PROGRAM MAIN
VAR
	
	// general use variables
	bLocalVar_1				: BOOL;
	bActivateTimeout		: BOOL;
	bHighLevelAlarm			: BOOL;
	bLowLevelAlarm			: BOOL;
	nRetryCounter			: USINT;
	tTotalCycleTime 		: TIME;
	tTimeoutTime			: TIME;
	sMachineState			: STRING(30);
	sPrevMachineState		: STRING(30);
	sErrorMsg				: STRING(50);
	tmrProcessTimer			: Tc2_Standard.TON;
	
	// function block and interface definitions
	fbFurnace 				: FB_Furnace;
	fbGantry 				: FB_Gantry;
	fbQuenchTank 			: FB_QuenchTank;
	fbRecipie				: FB_Recipe;
	fbAlarmManager			: FB_AlarmManager;
	fbTimeout				: FB_Timeout;
	fbStackLight			: FB_StackLight;
	iGantry					: I_Gantry;
	
	// recipe variables
	bCreateRecipe			: BOOL;
	bEditRecipe         	: BOOL;
	bDeleteRecipe			: BOOL;
	tHeatSetTime			: TIME;
	tQuenchTime				: TIME;
	sRecipeName				: STRING(20);
	
	// salt furnace variables
	bSaltCoverOn	    	: BOOL;	
	
	// quench tank variables

END_VAR

// *** GANTRY CONTROL ********************************************************************************

IF sMachineState = 'Startup' THEN
	sMachineState := 'Navigating Home';
	
ELSIF sMachineState = 'Idle' THEN
	sPrevMachineState := 'Idle';

ELSIF sMachineState = 'Navigating to Start Position' THEN
	IF sPrevMachineState <> 'Navigating to Start Position' THEN
		sPrevMachineState := 'Navigating to Start Position';
		iGantry.M_GoPreHeatSet();
		fbTimeout(bActivate := FALSE);
		bActivateTimeout := TRUE;
		tTimeoutTime := T#20S;
		nRetryCounter := 0;
	END_IF

	IF iGantry.M_GetPosition() = 'pre heat set' THEN
		sMachineState := 'Waiting for Start';
	ELSIF fbTimeout.nAttempts >= 3 THEN
		sMachineState := 'Help Required';
		sErrorMsg := 'Unable to move to start pos from home';
	ELSIF fbTimeout.nAttempts > nRetryCounter THEN
		iGantry.M_GoPreHeatSet();
		nRetryCounter := nRetryCounter + 1;
	END_IF

ELSIF sMachineState = 'Waiting for Start' THEN
    RETURN;
	
ELSIF sMachineState = 'Getting Salty' THEN
	IF sPrevMachineState <> 'Getting Salty' THEN
		sPrevMachineState := 'Getting Salty';
	    iGantry.M_GoHeatSet();
		fbTimeout(bActivate := FALSE);
		bActivateTimeout := TRUE;
		tTimeoutTime := T#10S;
		nRetryCounter := 0;
	END_IF

	IF iGantry.M_GetPosition() = 'setting shape' THEN
		sMachineState := 'Heat Soaking';
	ELSIF fbTimeout.nAttempts >= 3 THEN
		sMachineState := 'Help Required';
		sErrorMsg := 'Unable to enter salt bath';
	ELSIF fbTimeout.nAttempts > nRetryCounter THEN
		iGantry.M_GoHeatSet();
		nRetryCounter := nRetryCounter + 1;
	END_IF
	
ELSIF sMachineState = 'Heat Soaking' THEN
	IF sPrevMachineState <> 'Heat Soaking' THEN
		sPrevMachineState := 'Heat Soaking';
		tmrProcessTimer(IN := FALSE);
	END_IF
	
	tmrProcessTimer(IN := TRUE, PT := tHeatSetTime);
	IF tmrProcessTimer.Q THEN
		sMachineState := 'Navigating to Quench';
	END_IF
	
ELSIF sMachineState = 'Navigating to Quench' THEN
	IF sPrevMachineState <> 'Navigating to Quench' THEN
		sPrevMachineState := 'Navigating to Quench';
		iGantry.M_GoQuench();
		fbTimeout(bActivate := FALSE);
		bActivateTimeout := TRUE;
		tTimeoutTime := T#10S;
		nRetryCounter := 0;
	END_IF

	IF iGantry.M_GetPosition() = 'quenching' THEN
		sMachineState := 'Quenching';
	ELSIF fbTimeout.nAttempts >= 3 THEN
		sMachineState := 'Help Required';
		sErrorMsg := 'Unable to navigate from heat to quench';
	ELSIF fbTimeout.nAttempts > nRetryCounter THEN
		iGantry.M_GoHeatSet();
		nRetryCounter := nRetryCounter + 1;
	END_IF	

ELSIF sMachineState = 'Quenching' THEN
	IF sPrevMachineState <> 'Quenching' THEN
		sPrevMachineState := 'Quenching';
		tmrProcessTimer(IN := FALSE);
	END_IF
	
	tmrProcessTimer(IN := TRUE, PT := tQuenchTime);
	IF tmrProcessTimer.Q THEN
		sMachineState := 'Navigating Home';
	END_IF
	
ELSIF sMachineState = 'Navigating Home' THEN
	IF sPrevMachineState <> 'Navigating Home' THEN
		sPrevMachineState := 'Navigating Home';
		iGantry.M_GoHome();
		fbTimeout(bActivate := FALSE);
		bActivateTimeout := TRUE;
		tTimeoutTime := T#20S;
		nRetryCounter := 0;
	END_IF
	
	IF iGantry.M_GetPosition() = 'Home' THEN
		sMachineState := 'Idle';
	ELSIF fbTimeout.nAttempts >= 3 THEN
		sMachineState := 'Help Required';
		sErrorMsg := 'Unable to move to start pos from home';
	ELSIF fbTimeout.nAttempts > nRetryCounter THEN
		iGantry.M_GoPreHeatSet();
		nRetryCounter := nRetryCounter + 1;
	END_IF
	
END_IF

fbTimeout(bActivate := bActivateTimeout, tDuration := tTimeoutTime);


// *** RECIPE ACTIONS *********************************************************************************

IF bCreateRecipe THEN
	bCreateRecipe := FALSE;
	fbRecipie.M_Create(sName := sRecipeName, 
					   tIngredient_1 := tHeatSetTime, 
					   tIngredient_2 := tQuenchTime);
END_IF

IF bEditRecipe THEN
	bEditRecipe := FALSE;
	fbRecipie.M_Edit(sName := sRecipeName, 
					 tNewIngredient_1 := tHeatSetTime, 
					 tNewIngredient_2 := tQuenchTime);
END_IF

IF bDeleteRecipe THEN
	bDeleteRecipe := FALSE;
	fbRecipie.M_Delete(sName := sRecipeName);
END_IF


// *** QUENCH TANK OPERATION ***************************************************************************




// *** STACK LIGHT OPERATION ***************************************************************************

IF sMachineState = 'Idle' THEN
	IF bHighLevelAlarm THEN
		fbStackLight(bBlinkEnabled := FALSE, sColor := 'red');
	ELSIF bLowLevelAlarm THEN
		fbStackLight(bBlinkEnabled := FALSE, sColor := 'yellow');
	ELSE
		fbStackLight(bBlinkEnabled := FALSE, sColor := 'green');
	END_IF	
ELSE
	IF bHighLevelAlarm THEN
		fbStackLight(bBlinkEnabled := TRUE, sColor := 'red');
	ELSIF bLowLevelAlarm THEN
		fbStackLight(bBlinkEnabled := TRUE, sColor := 'yellow');
	ELSE
		fbStackLight(bBlinkEnabled := TRUE, sColor := 'green');
	END_IF	
END_IF

END_PROGRAM

(* stored: Version 1.1.0.1, ProductVersion 3.1.4024.11
   POU MAIN: Id {efa7bdf7-c0cf-482e-b1df-3f80349c525c}, SpecialFunc None *)
